TYPE csp_transfer_accumulator_connection_status_enum :
(		
	CSP_TRANSFER_ACCUMULATOR_STATUS_CONNECTION_START					:= 0,
	CSP_TRANSFER_ACCUMULATOR_STATUS_CONNECTION_ENGAGE					:= 10,
	CSP_TRANSFER_ACCUMULATOR_STATUS_CONNECTION_ENGAGED					:= 20,
	CSP_TRANSFER_ACCUMULATOR_STATUS_CONNECTION_CHECK_CHANGE_CAM			:= 30,
	CSP_TRANSFER_ACCUMULATOR_STATUS_CONNECTION_CHANGE_CAM				:= 40,
	CSP_TRANSFER_ACCUMULATOR_STATUS_CONNECTION_WAIT_NEW_CAM				:= 50,
	CSP_TRANSFER_ACCUMULATOR_STATUS_CONNECTION_DONE 					:= 900,
	CSP_TRANSFER_ACCUMULATOR_STATUS_CONNECTION_ERROR 					:= 999
) := CSP_TRANSFER_ACCUMULATOR_STATUS_CONNECTION_START;
END_TYPE

(* stored: Version 1.1.0.1, ProductVersion 3.1.4022.12
   DUT csp_transfer_accumulator_connection_status_enum: Id {f10c1315-aa02-451a-a38d-3a1cf2b32078} *)
